{attribute 'GeneratedUsingTerminal: EP2001-1000-0016'}
{attribute addProperty BoxType "EP2001-1000-0016"}
{attribute addProperty Id "Output5AT %Q*BOOL1Output6AT %Q*BOOL1Output7AT %Q*BOOL1Output8AT %Q*BOOL1"}
{attribute addProperty CRC "2412622741"}
{attribute addProperty Size "4"}
TYPE Group_8FCDB395 EXTENDS OutputBase_10CEE7DE :
STRUCT
	{attribute addProperty Name "Output5"}
	Output5 AT %Q* : BOOL;
	{attribute addProperty Name "Output6"}
	Output6 AT %Q* : BOOL;
	{attribute addProperty Name "Output7"}
	Output7 AT %Q* : BOOL;
	{attribute addProperty Name "Output8"}
	Output8 AT %Q* : BOOL;
END_STRUCT
END_TYPE

(* stored: Version 1.2.0.0, ProductVersion 3.1.4024.9
   DUT Group_8FCDB395: Id {a68f247f-2cad-463c-bcea-8c92f370b1b8} *)
